GLOBALCONSTANTS SubStrings (* Global constants *)
  (* Standard: 61499-1 *)
  (* Version 1.0, 2026-08-07, Franz Höpfinger, Meisterschulen am Ostbahnhof *)
  PACKAGE Meins::InputOutputTester::Button_OPC_UA;
  VAR_GLOBAL CONSTANT
    I1_WRITE : WSTRING := "opc_ua[WRITE;/Objects/DigitalInput/I1,1:s=I1]";
    I2_WRITE : WSTRING := "opc_ua[WRITE;/Objects/DigitalInput/I2,1:s=I2]";
    I3_WRITE : WSTRING := "opc_ua[WRITE;/Objects/DigitalInput/I3,1:s=I3]";
    I4_WRITE : WSTRING := "opc_ua[WRITE;/Objects/DigitalInput/I4,1:s=I4]";
    I5_WRITE : WSTRING := "opc_ua[WRITE;/Objects/DigitalInput/I5,1:s=I5]";
    I6_WRITE : WSTRING := "opc_ua[WRITE;/Objects/DigitalInput/I6,1:s=I6]";
    I7_WRITE : WSTRING := "opc_ua[WRITE;/Objects/DigitalInput/I7,1:s=I7]";
    I8_WRITE : WSTRING := "opc_ua[WRITE;/Objects/DigitalInput/I8,1:s=I8]";
    Q01_READ : WSTRING := "opc_ua[READ;/Objects/DigitalOutput/Q01,1:s=Q01]";
    Q01_WRITE : WSTRING := "opc_ua[WRITE;/Objects/DigitalOutput/Q01,1:s=Q01]";
    Q02_READ : WSTRING := "opc_ua[READ;/Objects/DigitalOutput/Q02,1:s=Q02]";
    Q02_WRITE : WSTRING := "opc_ua[WRITE;/Objects/DigitalOutput/Q02,1:s=Q02]";
    Q03_READ : WSTRING := "opc_ua[READ;/Objects/DigitalOutput/Q03,1:s=Q03]";
    Q03_WRITE : WSTRING := "opc_ua[WRITE;/Objects/DigitalOutput/Q03,1:s=Q03]";
    Q04_READ : WSTRING := "opc_ua[READ;/Objects/DigitalOutput/Q04,1:s=Q04]";
    Q04_WRITE : WSTRING := "opc_ua[WRITE;/Objects/DigitalOutput/Q04,1:s=Q04]";
    Q05_READ : WSTRING := "opc_ua[READ;/Objects/DigitalOutput/Q05,1:s=Q05]";
    Q05_WRITE : WSTRING := "opc_ua[WRITE;/Objects/DigitalOutput/Q05,1:s=Q05]";
    Q06_READ : WSTRING := "opc_ua[READ;/Objects/DigitalOutput/Q06,1:s=Q06]";
    Q06_WRITE : WSTRING := "opc_ua[WRITE;/Objects/DigitalOutput/Q06,1:s=Q06]";
    Q07_READ : WSTRING := "opc_ua[READ;/Objects/DigitalOutput/Q07,1:s=Q07]";
    Q07_WRITE : WSTRING := "opc_ua[WRITE;/Objects/DigitalOutput/Q07,1:s=Q07]";
    Q08_READ : WSTRING := "opc_ua[READ;/Objects/DigitalOutput/Q08,1:s=Q08]";
    Q08_WRITE : WSTRING := "opc_ua[WRITE;/Objects/DigitalOutput/Q08,1:s=Q08]";
    Q09_READ : WSTRING := "opc_ua[READ;/Objects/DigitalOutput/Q09,1:s=Q09]";
    Q09_WRITE : WSTRING := "opc_ua[WRITE;/Objects/DigitalOutput/Q09,1:s=Q09]";
    Q10_READ : WSTRING := "opc_ua[READ;/Objects/DigitalOutput/Q10,1:s=Q10]";
    Q10_WRITE : WSTRING := "opc_ua[WRITE;/Objects/DigitalOutput/Q10,1:s=Q10]";
    Q11_READ : WSTRING := "opc_ua[READ;/Objects/DigitalOutput/Q11,1:s=Q11]";
    Q11_WRITE : WSTRING := "opc_ua[WRITE;/Objects/DigitalOutput/Q11,1:s=Q11]";
    Q12_READ : WSTRING := "opc_ua[READ;/Objects/DigitalOutput/Q12,1:s=Q12]";
    Q12_WRITE : WSTRING := "opc_ua[WRITE;/Objects/DigitalOutput/Q12,1:s=Q12]";
    Tick_WRITE : WSTRING := "opc_ua[WRITE;/Objects/System/Tick,1:s=System.Tick]";
  END_VAR
END_GLOBALCONSTANTS
